TYPE ST_CylinderInputs :
STRUCT
	fPistonPressure : INT;
	fRodPressure : INT; 
	fCylinderPosition : LREAL; 
END_STRUCT
END_TYPE

(* stored: Version 1.1.0.1, ProductVersion 3.1.4024.12
   DUT ST_CylinderInputs: Id {d2edb17a-f020-4013-b394-0449d935e4b1} *)
